TYPE T_EX260MEC1_ValveList : USINT; END_TYPE

(* stored: Version 1.1.0.1, ProductVersion 3.1.4024.16
   DUT T_EX260MEC1_ValveList: Id {3a8b2d86-7c7a-07c6-159f-0d84bd6aa22c} *)
